(* CODESYS project pluginbeckhoffethercatasycube.library
   Author: Asyril SA
   Placeholder: Plugin Ethercat Asycube
   Title: Plugin Ethercat Asycube
   Version: 1.1.0
   Description: This library is created for controling the Asycube product
   Company: Asyril SA

Project tree, tasks and I/O mapping:
  libraries: Tc2_Standard, * (Beckhoff Automation GmbH); Tc2_System, * (Beckhoff Automation GmbH); Tc2_Utilities, * (Beckhoff Automation GmbH); Tc3_Module, * (Beckhoff Automation GmbH); VisuDialogs, * (System); VisuSymbols, 3.5.10.0 (System)
  DUTs/
    data type asycubeReadHoldingRegister
    data type asycubeWriteHoldingRegister
    data type HOLDING_REGISTERS_READ
    data type HOLDING_REGISTERS_WRITE
  GVLs/
    global variables dbGateway
  POUs/
    function block FB_Backlight [ST]
    function block FB_Execute_Hopper_Vibration [ST]
    function block FB_Execute_Platform_Vibration [ST]
    function block FB_Execute_Sequence [ST]
    program MAIN [FBD]
  VISUs/
  text list GlobalTextList
*)

// DUTs/asycubeReadHoldingRegister
TYPE asycubeReadHoldingRegister :
UNION
	w				: INT;
	b 		AT %I* 	: ARRAY[0..1] OF BYTE;
END_UNION
END_TYPE

// DUTs/asycubeWriteHoldingRegister
TYPE asycubeWriteHoldingRegister :
UNION
	w				: INT;
	b 		AT %Q* 	: ARRAY[0..1] OF BYTE;
END_UNION
END_TYPE

// DUTs/HOLDING_REGISTERS_READ
TYPE HOLDING_REGISTERS_READ :
STRUCT
	HR_MODBUS_STATUS: asycubeReadHoldingRegister;
	HR_MODBUS_ERROR_CODE: asycubeReadHoldingRegister;
	HR_WARNINGS: asycubeReadHoldingRegister;
	HR_ALARMS: asycubeReadHoldingRegister;
	HR_MODBUS_PLATFORM_STATUS: asycubeReadHoldingRegister;
	HR_PLATFORM_REMAINING_TIME: asycubeReadHoldingRegister;
	HR_MODBUS_HOPPER_STATUS: asycubeReadHoldingRegister;
	HR_HOPPER_REMAINING_TIME: asycubeReadHoldingRegister;
	HR_MODBUS_SEQUENCE_STATUS: asycubeReadHoldingRegister;
	HR_SEQUENCE_REMAINING_TIME: asycubeReadHoldingRegister;
	HR_VIBRATION_SET_SELECTED: asycubeReadHoldingRegister;
	HR_SEQUENCE_SELECTED: asycubeReadHoldingRegister;
	HR_BACKLIGHT_STATE_STATUS: asycubeReadHoldingRegister;
	HR_READ_WRITE_PARAMETER_READ_VALUE: asycubeReadHoldingRegister;
	HR_FIRMWARE_VERSION_H: asycubeReadHoldingRegister;
	HR_FIRMWARE_VERSION_M: asycubeReadHoldingRegister;
	HR_FIRMWARE_VERSION_L: asycubeReadHoldingRegister;
	HR_USER_ACCESS_LEVEL: asycubeReadHoldingRegister;
	HR_FLASH_OPERATIONS_STATUS: asycubeReadHoldingRegister;
	HR_MODBUS_COMMUNICATION_STATUS_L: asycubeReadHoldingRegister;
	HR_MODBUS_COMMUNICATION_STATUS_H: asycubeReadHoldingRegister;
	HR_ETHERCAT_COMMUNICATION_STATUS: asycubeReadHoldingRegister;

END_STRUCT
END_TYPE

// DUTs/HOLDING_REGISTERS_WRITE
TYPE HOLDING_REGISTERS_WRITE :
STRUCT
	HR_MODBUS_CONTROL: asycubeWriteHoldingRegister;
	HR_PLATFORM_VIBRATION_TRIG: asycubeWriteHoldingRegister;
	HR_PLATFORM_VIBRATION_ID: asycubeWriteHoldingRegister;
	HR_PLATFORM_VIBRATION_DURATION: asycubeWriteHoldingRegister;
	HR_PLATFORM_CENTERING_TRIG: asycubeWriteHoldingRegister;
	HR_PLATFORM_CENTERING_X: asycubeWriteHoldingRegister;
	HR_PLATFORM_CENTERING_Y: asycubeWriteHoldingRegister;
	HR_HOPPER_VIBRATION_TRIG: asycubeWriteHoldingRegister;
	HR_HOPPER_VIBRATION_ID: asycubeWriteHoldingRegister;
	HR_HOPPER_VIBRATION_DURATION: asycubeWriteHoldingRegister;
	HR_HOPPER_FEEDING_TRIG: asycubeWriteHoldingRegister;
	HR_HOPPER_FEEDING_VIBRATION: asycubeWriteHoldingRegister;
	HR_HOPPER_FEEDING_NBPARTS: asycubeWriteHoldingRegister;
	HR_HOPPER_FEEDING_NBMAX: asycubeWriteHoldingRegister;
	HR_SEQUENCE_EXECUTION_TRIG: asycubeWriteHoldingRegister;
	HR_SEQUENCE_EXECUTION_NBPARTS: asycubeWriteHoldingRegister;
	HR_SEQUENCE_EXECUTION_NBMAX: asycubeWriteHoldingRegister;
	HR_SEQUENCE_EXECUTION_X: asycubeWriteHoldingRegister;
	HR_SEQUENCE_EXECUTION_Y: asycubeWriteHoldingRegister;
	HR_SEQUENCE_EXECUTION_SEQUENCEID: asycubeWriteHoldingRegister;
	HR_SELECT_VIBRATION_SET: asycubeWriteHoldingRegister;
	HR_SELECT_SEQUENCE: asycubeWriteHoldingRegister;
	HR_BACKLIGHT_STATE_CONTROL: asycubeWriteHoldingRegister;
	HR_EXECUTE_BACKLIGHT_FLASH_TRIG: asycubeWriteHoldingRegister;
	HR_BACKLIGHT_INTENSITY_TRIG: asycubeWriteHoldingRegister;
	HR_BACKLIGHT_INTENSITY: asycubeWriteHoldingRegister;
	HR_PLATFORM_HALT: asycubeWriteHoldingRegister;
	HR_HOPPER_HALT: asycubeWriteHoldingRegister;
	HR_SEQUENCE_HALT: asycubeWriteHoldingRegister;
	HR_READ_WRITE_PARAMETER_TRIG: asycubeWriteHoldingRegister;
	HR_READ_WRITE_PARAMETER_ADDRESS: asycubeWriteHoldingRegister;
	HR_READ_WRITE_PARAMETER_WRITE_VALUE: asycubeWriteHoldingRegister;
	HR_FLASH_OPERATIONS: asycubeWriteHoldingRegister;
	
END_STRUCT
END_TYPE

// GVLs/dbGateway
{attribute 'qualified_only'}
VAR_GLOBAL
	regAsycubeRead			: HOLDING_REGISTERS_READ;		//Register for read in Asycube
	regAsycubeWrite			: HOLDING_REGISTERS_WRITE;		//Register for write in Asycube
	
END_VAR

// POUs/FB_Backlight
FUNCTION_BLOCK FB_Backlight
VAR_INPUT
	{attribute 'pingroup' := 'Working'}
	boLightONPIN				: BOOL;							//Turn ON the Backlight
	{attribute 'pingroup' := 'Working'}
	boLightOFFPIN				: BOOL;							//Turn OFF the Backlight
	{attribute 'pingroup' := 'Working'}
	tiDurationPIN				: TIME;							//Duration of backlight
	
END_VAR
VAR_IN_OUT					
	{attribute 'pingroup' := 'Gateway'}
	regAsycubeWritePIO			: HOLDING_REGISTERS_WRITE;		//Register for writing to Asycube
	{attribute 'pingroup' := 'Gateway'}
	regAsycubeReadPIO			: HOLDING_REGISTERS_READ;		//Register for reading to Asycube
	
END_VAR
VAR_OUTPUT
	{attribute 'pingroup' := 'Working'}
	woStatePOU					: WORD;							//0 = IDLE, 1 = Running, 2 = Stopping, 10 = Error
	{attribute 'pingroup' := 'Working'}
	tiRemainingTimePOU			: TIME;							//Time remaining of backlight
	
	{attribute 'pingroup' := 'Error Management'}
	boErrorPOU					: BOOL;							//Error
	{attribute 'pingroup' := 'Error Management'}
	inErrorIDPOU				: INT;							//Error ID
	{attribute 'pingroup' := 'Error Management'}
	stErrorNamePOU				: STRING;						//Name of error
	
END_VAR
VAR
	R_TRIG_Start				: R_TRIG;						//Rising edge of start
	R_TRIG_Stop					: R_TRIG;						//Rising edge of stop
	TOF_Duration				: TOF;							//Duration of backlight
	R_TRIG_State1				: R_TRIG;						//Rising edge of number sequence 1
	TON_TimeOut					: TON;							//Temporisation of time out communication
	
	woLastStateLST				: WORD;							//Last state
	boErrorTransitionLST		: BOOL;							//Error transition
	boErrorTimeOutLST			: BOOL;							//Error time out
	boErrorComAsycubeLST		: BOOL;							//Error communication Asycube
	boErrorComGatewayLST		: BOOL;							//Error communication gateway
END_VAR

//=============================================================================
// Asyril SA
// (c)Copyright 2019 
//-----------------------------------------------------------------------------
// Library:       Plugin Asycube EtherCat Beckhoff   
// Tested with:   C6015
// Engineering:   Twincat 3.1.4024.7
// Restrictions:  -
// Requirements:  -
// Functionality: FB_Backlight, Management of asycube backlight.
//-----------------------------------------------------------------------------
// Change log table:
// Version  Date       In charge / Changes applied
// 1.0      26.03.2020 DcA         Version inital.
// 1.1 		23.09.2020 DcA		   Added precision in connection errors.
// 
//=============================================================================

//Declarations of program instances (trigger and temporisation)
{region "Trigger"}

//Rising trigger of light on
R_TRIG_Start(CLK:= boLightONPIN);

//Rising trigger of light off
R_TRIG_Stop(CLK:= boLightOFFPIN);

//Rising trigger of running state
R_TRIG_State1(CLK:= woStatePOU = 1);

//Temporisation of light on
TOF_Duration(IN:= R_TRIG_State1.Q, PT:= tiDurationPIN);

//Temporisation of time out of communication
TON_TimeOut(IN:= (woStatePOU = 1 AND regAsycubeReadPIO.HR_BACKLIGHT_STATE_STATUS.w = 0)
				OR (woStatePOU = 0 AND regAsycubeReadPIO.HR_BACKLIGHT_STATE_STATUS.w = 1), PT:= T#5S);
	
//Initialisation
tiRemainingTimePOU := T#0S;		 
	 
{endregion}
	 
	 
//Region of working programm
{region "Working"}

//Sequence state diagram
CASE woStatePOU OF
	
	0:	//IDLE
	
	IF boErrorPOU THEN
		woStatePOU := 10;
	ELSIF R_TRIG_Start.Q THEN
		woStatePOU := 1;
	END_IF;
	
	1:	//Running
	
	IF boErrorPOU THEN
		woStatePOU := 10;
	ELSIF R_TRIG_Start.Q THEN
		woStatePOU := 10;
		boErrorTransitionLST := TRUE;
	ELSIF R_TRIG_Stop.Q OR (TOF_Duration.ET >= tiDurationPIN AND tiDurationPIN > T#0MS) THEN
		woStatePOU := 2;
	END_IF;
	
	2:	//Stopping
	
	IF boErrorPOU THEN
		woStatePOU := 10;
	ELSIF R_TRIG_Start.Q THEN
		woStatePOU := 10; 
		boErrorTransitionLST := TRUE;
	ELSIF regAsycubeReadPIO.HR_BACKLIGHT_STATE_STATUS.w = 0 THEN
		woStatePOU := 0;
	END_IF;
	
	10:	//Error

	IF NOT boErrorPOU THEN
		woStatePOU := 2;
	END_IF;

END_CASE;

//Parameters processing

//If it is in running
IF woStatePOU = 1 THEN
	regAsycubeWritePIO.HR_BACKLIGHT_STATE_CONTROL.w := 1;
	tiRemainingTimePOU := tiDurationPIN - TOF_Duration.ET;
END_IF;

//If it is in stopping
IF woStatePOU = 2 THEN
	regAsycubeWritePIO.HR_BACKLIGHT_STATE_CONTROL.w := 0;
	regAsycubeWritePIO.HR_MODBUS_CONTROL.w := 16#00;
END_IF;

//If it is in error
IF woStatePOU = 10 THEN
	regAsycubeWritePIO.HR_BACKLIGHT_STATE_CONTROL.w := 0;
END_IF;

//Save last state before error state
IF woStatePOU <> 10 THEN
	woLastStateLST := woStatePOU;
END_IF;

//If it is in error (trigger)
IF (R_TRIG_Stop.Q AND woStatePOU = 10) OR 
	((regAsycubeReadPIO.HR_MODBUS_COMMUNICATION_STATUS_L.w = 4 AND regAsycubeReadPIO.HR_ETHERCAT_COMMUNICATION_STATUS.w = 8) AND 
	(boErrorComAsycubeLST OR boErrorComGatewayLST) AND 
	woLastStateLST = 0) THEN
	
	regAsycubeWritePIO.HR_MODBUS_CONTROL.w := 16#FF;
	boErrorTransitionLST := FALSE;
	boErrorComAsycubeLST := FALSE;
	boErrorComGatewayLST := FALSE;
	boErrorTimeOutLST := FALSE;
END_IF;
	 
{endregion}

//Management of error
{region "Error"}
	
//Time out communciation	
IF TON_TimeOut.Q THEN
	boErrorTimeOutLST := TRUE;
END_IF;

//Asycube disconnected
IF regAsycubeReadPIO.HR_MODBUS_COMMUNICATION_STATUS_L.w <> 4 AND woStatePOU <> 10 THEN
	boErrorComAsycubeLST := TRUE;
END_IF;

//Gateway disconnected
IF regAsycubeReadPIO.HR_ETHERCAT_COMMUNICATION_STATUS.w <> 8 AND woStatePOU <> 10 THEN
	boErrorComGatewayLST := TRUE;
END_IF;
  
//If an error is active
IF	((regAsycubeReadPIO.HR_MODBUS_STATUS.w <> 0 OR boErrorTransitionLST) AND woStatePOU <> 0) OR 
	boErrorTimeOutLST OR boErrorComAsycubeLST OR boErrorComGatewayLST THEN
		 
	boErrorPOU := TRUE;
			
		//Error transition
		IF boErrorTransitionLST THEN
			inErrorIDPOU := 730;
			stErrorNamePOU := 'Transition Error';
		//Asycube  Modbus  errors  status
		ELSIF (INT_TO_UINT(regAsycubeReadPIO.HR_MODBUS_STATUS.w) AND 16#01) = 16#01 THEN	
			inErrorIDPOU := 731;	
	  		stErrorNamePOU := 'Asycube Modbus Error : 0x';
			stErrorNamePOU := CONCAT(STR1:= stErrorNamePOU, STR2:= DWORD_TO_HEXSTR( UINT_TO_DWORD( INT_TO_UINT(regAsycubeReadPIO.HR_MODBUS_ERROR_CODE.w) AND 16#00FF ), 4, FALSE ) ); 
				 
		//Internal  Modbus  communication  errorstatus
		ELSIF (INT_TO_UINT(regAsycubeReadPIO.HR_MODBUS_STATUS.w) AND 16#02) = 16#02 THEN
			inErrorIDPOU := 732;
			stErrorNamePOU := 'Asycube Internal Modbus Error : 0x';
			stErrorNamePOU := CONCAT(STR1:= stErrorNamePOU, STR2:= DWORD_TO_HEXSTR( UINT_TO_DWORD( SHL( INT_TO_UINT(regAsycubeReadPIO.HR_MODBUS_ERROR_CODE.w) AND 16#FF00 , 2) ) , 4, FALSE ) ); 
						   
		//Asycube  warnings  status
		ELSIF (INT_TO_UINT(regAsycubeReadPIO.HR_MODBUS_STATUS.w) AND 16#04) = 16#04 THEN
			inErrorIDPOU := 733;
			stErrorNamePOU := 'Asycube Warnings : 0x';
			stErrorNamePOU := CONCAT(STR1:= stErrorNamePOU, STR2:= DWORD_TO_HEXSTR( INT_TO_DWORD(regAsycubeReadPIO.HR_WARNINGS.w), 4, FALSE ) ); 

		//Asycube alarms status
		ELSIF (INT_TO_UINT(regAsycubeReadPIO.HR_MODBUS_STATUS.w) AND 16#08) = 16#08 THEN
			inErrorIDPOU := 734;
			stErrorNamePOU := 'Asycube Alarms : 0x';
			stErrorNamePOU := CONCAT(STR1:= stErrorNamePOU, STR2:= DWORD_TO_HEXSTR( INT_TO_DWORD(regAsycubeReadPIO.HR_ALARMS.w), 4, FALSE ) );   	
 
		//Gateway disconnected from plc
		ELSIF boErrorComGatewayLST THEN
			inErrorIDPOU := 735;
			stErrorNamePOU := 'Gateway disconnected from PLC';
		
		//Asycube disconnected from gateway
		ELSIF boErrorComAsycubeLST THEN
			inErrorIDPOU := 736;
			stErrorNamePOU := 'Asycube disconnected from gateway';
		
		//Communication time out
		ELSIF boErrorTimeOutLST THEN
			inErrorIDPOU := 737;
			stErrorNamePOU := 'Time out';

	 	//Unknown error
		ELSE 
			inErrorIDPOU := 739;
			stErrorNamePOU := 'N/A';
		END_IF;  

ELSE
	boErrorPOU := FALSE;
	inErrorIDPOU := 0;
	stErrorNamePOU := '';	 
END_IF;
	 
{endregion}

END_FUNCTION_BLOCK

// POUs/FB_Execute_Hopper_Vibration
FUNCTION_BLOCK FB_Execute_Hopper_Vibration
VAR_INPUT
	{attribute 'pingroup' := 'Working'}
	inSelectModePIN				: INT;							//0 = Vibration, 1 = Hopping
	{attribute 'pingroup' := 'Working'}
	boStartPIN					: BOOL;							//Start vibration
	{attribute 'pingroup' := 'Working'}
	boStopPIN					: BOOL;							//Stop vibration
	{attribute 'pingroup' := 'Working'}
	inVibrationIDPIN			: INT:=0;						//Vibration ID (0..25)
	{attribute 'pingroup' := 'Working'}
	inVibrationSetPIN			: INT:=1;						//Vibration Set (1..26)
	{attribute 'pingroup' := 'Working'}
	inNbPartsPIN				: INT;							//Number of parts on the cube
	{attribute 'pingroup' := 'Working'}
	inNbPartsMaxPIN				: INT;							//Number max of parts on the cube
	{attribute 'pingroup' := 'Working'}
	tiDurationPIN				: TIME;							//Time duration of vibration

END_VAR
VAR_IN_OUT
	{attribute 'pingroup' := 'Gateway'}
	regAsycubeWritePIO			: HOLDING_REGISTERS_WRITE;		//Register for writing to Asycube
	{attribute 'pingroup' := 'Gateway'}
	regAsycubeReadPIO			: HOLDING_REGISTERS_READ;		//Register for reading to Asycube
	
END_VAR
VAR_OUTPUT
	{attribute 'pingroup' := 'Working'}
	woStatePOU					: WORD;							//0 = IDLE, 1 = Running, 2 = Stopping, 10 = Error
	{attribute 'pingroup' := 'Working'}
	boDonePOU					: BOOL;							//Vibration is done
	{attribute 'pingroup' := 'Working'}
	tiRemainingTimePOU			: TIME;							//Time remaining of vibration
	
	{attribute 'pingroup' := 'Error Management'}
	boErrorPOU					: BOOL;							//Error
	{attribute 'pingroup' := 'Error Management'}
	inErrorIDPOU				: INT;							//Error ID
	{attribute 'pingroup' := 'Error Management'}
	stErrorNamePOU				: STRING;						//Name of error
	

END_VAR
VAR
	R_TRIG_Start				: R_TRIG;						//Rising edge of start
	R_TRIG_Stop					: R_TRIG;						//Rising edge of stop
	R_TRIG_State1				: R_TRIG;						//Rising edge step number 1
	R_TRIG_Done					: R_TRIG;						//Rising edge of vibration done 
	TON_TimeOut					: TON;							//Temporisation of time out communication
	
	woLastStateLST				: WORD;							//Last state
	boErrorTransitionLST		: BOOL;							//Error transition
	boErrorTimeOutLST			: BOOL;							//Error time out
	boErrorComAsycubeLST		: BOOL;							//Error communication Asycube
	boErrorComGatewayLST		: BOOL;							//Error communication gateway
	boErrorParameterLST			: BOOL;							//Error parameters
	
END_VAR

//=============================================================================
// Asyril SA
// (c)Copyright 2019 
//-----------------------------------------------------------------------------
// Library:       Plugin Asycube EtherCat Beckhoff   
// Tested with:   C6015
// Engineering:   Twincat 3.1.4024.7
// Restrictions:  -
// Requirements:  -
// Functionality: FB_Execute_Hopper_Vibration, Management of hopper vibration.
//-----------------------------------------------------------------------------
// Change log table:
// Version  Date       In charge / Changes applied
// 1.0      26.03.2020 DcA         Version initale.
// 1.1 		23.09.2020 DcA		   Added precision in connection errors.
// 
//=============================================================================

//Declarations of program instances (trigger and temporisation)
{region "Trigger"}

//Rising trigger of start
R_TRIG_Start(CLK:= boStartPIN);

//Rising trigger of stop
R_TRIG_Stop(CLK:= boStopPIN);

//Rising trigger of running state
R_TRIG_State1(CLK:= woStatePOU = 1);

//Rising trigger of vibration done
R_TRIG_Done(CLK:= regAsycubeReadPIO.HR_MODBUS_HOPPER_STATUS.w = 0);
	 
//Temporisation of time out of communication
TON_TimeOut(IN:= (woStatePOU = 1 AND regAsycubeReadPIO.HR_MODBUS_HOPPER_STATUS.w = 0)
				OR (woStatePOU = 0 AND regAsycubeReadPIO.HR_MODBUS_HOPPER_STATUS.w = 1), PT:= T#5S);
		  
{endregion}
	 
//Region of working programm
{region "Working"}

//Sequence state diagram
CASE woStatePOU OF
	
	0:	//IDLE
		 
	IF boErrorPOU THEN
		woStatePOU := 10;
		boDonePOU := FALSE;
	ELSIF R_TRIG_Start.Q THEN
		woStatePOU := 1;
		boDonePOU := FALSE;
	END_IF;
	
	1:	//Running

	IF boErrorPOU THEN
		woStatePOU := 10;
	ELSIF R_TRIG_Start.Q THEN
		woStatePOU := 10;
		boErrorTransitionLST := TRUE;
	ELSIF R_TRIG_Stop.Q THEN
		woStatePOU := 2;
	ELSIF R_TRIG_Done.Q THEN
		woStatePOU := 2;
		boDonePOU := TRUE;
	END_IF;
	
	2:	//Stopping

	IF boErrorPOU THEN
		woStatePOU := 10;
	ELSIF R_TRIG_Start.Q THEN
		woStatePOU := 10;
		boErrorTransitionLST := TRUE;
	ELSIF regAsycubeReadPIO.HR_MODBUS_HOPPER_STATUS.w = 0 THEN
		woStatePOU := 0;
	END_IF;
	
	10:	//Error

	IF NOT boErrorPOU THEN
		woStatePOU := 2;
	END_IF;

END_CASE;

//Parameters processing

//If it is in IDLE
IF woStatePOU = 0 THEN
	regAsycubeWritePIO.HR_HOPPER_HALT.w := 0;
END_IF;

//If it is in running (trigger) and vibration mode
IF R_TRIG_State1.Q AND inSelectModePIN = 0 THEN
	regAsycubeWritePIO.HR_HOPPER_VIBRATION_TRIG.w := 1;
END_IF;

//If it is in running (trigger) and feeding mode
IF R_TRIG_State1.Q AND inSelectModePIN = 1 THEN
	regAsycubeWritePIO.HR_HOPPER_FEEDING_TRIG.w := 1;
END_IF;

//If it is in running
IF inSelectModePIN = 0 AND tiDurationPIN = T#0MS THEN
	tiRemainingTimePOU := T#0S;
ELSE
	tiRemainingTimePOU := INT_TO_TIME(regAsycubeReadPIO.HR_HOPPER_REMAINING_TIME.w);
END_IF;

//If it is in stopping
IF woStatePOU = 2 THEN
	regAsycubeWritePIO.HR_HOPPER_VIBRATION_TRIG.w := 0;
	regAsycubeWritePIO.HR_HOPPER_FEEDING_TRIG.w := 0;
	regAsycubeWritePIO.HR_HOPPER_HALT.w := 1;
	regAsycubeWritePIO.HR_MODBUS_CONTROL.w := 16#00;
END_IF;

//If it is in error
IF woStatePOU = 10 THEN
	regAsycubeWritePIO.HR_HOPPER_VIBRATION_TRIG.w := 0;
	regAsycubeWritePIO.HR_HOPPER_FEEDING_TRIG.w := 0;
	regAsycubeWritePIO.HR_HOPPER_HALT.w := 1;
END_IF;
		  
//Save last state before error state
IF woStatePOU <> 10 THEN
	woLastStateLST := woStatePOU;
END_IF;

//If it is in error (trigger)
IF (R_TRIG_Stop.Q AND woStatePOU = 10) OR 
	((regAsycubeReadPIO.HR_MODBUS_COMMUNICATION_STATUS_L.w = 4 AND regAsycubeReadPIO.HR_ETHERCAT_COMMUNICATION_STATUS.w = 8) AND 
	(boErrorComAsycubeLST OR boErrorComGatewayLST) AND 
	woLastStateLST = 0) THEN
	
	regAsycubeWritePIO.HR_MODBUS_CONTROL.w := 16#FF;
	boErrorTransitionLST := FALSE;
	boErrorTimeOutLST := FALSE;
	boErrorComAsycubeLST := FALSE;
	boErrorComGatewayLST := FALSE;
	boErrorParameterLST := FALSE;
END_IF;

//Set parameters
//Position and duration paramater
regAsycubeWritePIO.HR_HOPPER_VIBRATION_DURATION.w := TIME_TO_INT(tiDurationPIN);
regAsycubeWritePIO.HR_HOPPER_FEEDING_NBMAX.w := inNbPartsMaxPIN;
regAsycubeWritePIO.HR_HOPPER_FEEDING_NBPARTS.w := inNbPartsPIN;

//Vibration ID parameter
IF inVibrationIDPIN > 25 AND woStatePOU = 1 THEN
	boErrorParameterLST := TRUE;
ELSIF inVibrationIDPIN < 0 AND woStatePOU = 1 THEN
	boErrorParameterLST := TRUE;
ELSIF woStatePOU = 1 THEN
	regAsycubeWritePIO.HR_HOPPER_VIBRATION_ID.w := inVibrationIDPIN;
	regAsycubeWritePIO.HR_HOPPER_FEEDING_VIBRATION.w := inVibrationIDPIN;
END_IF;

//Vibration set parameter  
IF inVibrationSetPIN > 26 AND woStatePOU = 1 THEN
	boErrorParameterLST := TRUE;
ELSIF inVibrationSetPIN < 1 AND woStatePOU = 1 THEN
	boErrorParameterLST := TRUE;
ELSIF woStatePOU = 1 THEN
	regAsycubeWritePIO.HR_SELECT_VIBRATION_SET.w := inVibrationSetPIN;
END_IF;

{endregion}

//Reion Error management
{region "Error"}

//Time out communication
IF TON_TimeOut.Q THEN
	boErrorTimeOutLST := TRUE;
END_IF;

//Asycube disconnected
IF regAsycubeReadPIO.HR_MODBUS_COMMUNICATION_STATUS_L.w <> 4 AND woStatePOU <> 10 THEN
	boErrorComAsycubeLST := TRUE;
END_IF;

//Gateway disconnected
IF regAsycubeReadPIO.HR_ETHERCAT_COMMUNICATION_STATUS.w <> 8 AND woStatePOU <> 10 THEN
	boErrorComGatewayLST := TRUE;
END_IF;

//If an error is active
IF	((regAsycubeReadPIO.HR_MODBUS_STATUS.w <> 0 OR boErrorTransitionLST OR boErrorParameterLST) AND woStatePOU <> 0) OR 
	boErrorTimeOutLST OR boErrorComAsycubeLST OR 
	boErrorComGatewayLST OR regAsycubeReadPIO.HR_MODBUS_HOPPER_STATUS.w = 2 THEN
	
	boErrorPOU := TRUE;
			
		//Error transition
		IF boErrorTransitionLST THEN
			inErrorIDPOU := 720;
			stErrorNamePOU := 'Transition Error';
		//Asycube  Modbus  errors  status
		ELSIF (INT_TO_UINT(regAsycubeReadPIO.HR_MODBUS_STATUS.w) AND 16#01) = 16#01 THEN	
			inErrorIDPOU := 721;	
	  		stErrorNamePOU := 'Asycube Modbus Error : 0x';
			stErrorNamePOU := CONCAT(STR1:= stErrorNamePOU, STR2:= DWORD_TO_HEXSTR( UINT_TO_DWORD( INT_TO_UINT(regAsycubeReadPIO.HR_MODBUS_ERROR_CODE.w) AND 16#00FF ), 4, FALSE ) ); 
				 
		//Internal  Modbus  communication  errorstatus
		ELSIF (INT_TO_UINT(regAsycubeReadPIO.HR_MODBUS_STATUS.w) AND 16#02) = 16#02 THEN
			inErrorIDPOU := 722;
			stErrorNamePOU := 'Asycube Internal Modbus Error : 0x';
			stErrorNamePOU := CONCAT(STR1:= stErrorNamePOU, STR2:= DWORD_TO_HEXSTR( UINT_TO_DWORD( SHL( INT_TO_UINT(regAsycubeReadPIO.HR_MODBUS_ERROR_CODE.w) AND 16#FF00 , 2) ) , 4, FALSE ) ); 
						   
		//Asycube  warnings  status
		ELSIF (INT_TO_UINT(regAsycubeReadPIO.HR_MODBUS_STATUS.w) AND 16#04) = 16#04 THEN
			inErrorIDPOU := 723;
			stErrorNamePOU := 'Asycube Warnings : 0x';
			stErrorNamePOU := CONCAT(STR1:= stErrorNamePOU, STR2:= DWORD_TO_HEXSTR( INT_TO_DWORD(regAsycubeReadPIO.HR_WARNINGS.w), 4, FALSE ) ); 

		//Asycube alarms status
		ELSIF (INT_TO_UINT(regAsycubeReadPIO.HR_MODBUS_STATUS.w) AND 16#08) = 16#08 THEN
			inErrorIDPOU := 724;
			stErrorNamePOU := 'Asycube Alarms : 0x';
			stErrorNamePOU := CONCAT(STR1:= stErrorNamePOU, STR2:= DWORD_TO_HEXSTR( INT_TO_DWORD(regAsycubeReadPIO.HR_ALARMS.w), 4, FALSE ) );   	
 
		//Gateway disconnected from plc
		ELSIF boErrorComGatewayLST THEN
			inErrorIDPOU := 725;
			stErrorNamePOU := 'Gateway disconnected from PLC';
		
		//Asycube disconnected from gateway
		ELSIF boErrorComAsycubeLST THEN
			inErrorIDPOU := 726;
			stErrorNamePOU := 'Asycube disconnected from gateway';
		
		//Communication time out
		ELSIF boErrorTimeOutLST THEN
			inErrorIDPOU := 727;
			stErrorNamePOU := 'Time out';
			 
		//Incorrect parameters
		ELSIF boErrorParameterLST THEN
			inErrorIDPOU := 728;
			stErrorNamePOU := 'Wrong parameter';
			//See variable error
			IF inVibrationIDPIN > 26 OR inVibrationIDPIN < 1 THEN
				stErrorNamePOU := CONCAT(stErrorNamePOU , ' : inVibrationIDPIN' );
			ELSIF inVibrationSetPIN > 26 OR inVibrationSetPIN < 1 THEN
				stErrorNamePOU := CONCAT(stErrorNamePOU , ' : inVibrationSetPIN' );
			END_IF;
				 
		//Unknown error
		ELSE 
			inErrorIDPOU := 729;
			stErrorNamePOU := 'N/A';
		END_IF;  

ELSE
	boErrorPOU := FALSE;
	inErrorIDPOU := 0;
	stErrorNamePOU := '';	 
END_IF;
	 
{endregion}

END_FUNCTION_BLOCK

// POUs/FB_Execute_Platform_Vibration
FUNCTION_BLOCK FB_Execute_Platform_Vibration
VAR_INPUT
	{attribute 'pingroup' := 'Working'}
	inSelectModePIN				: INT;							//0 = Vibration, 1 = Centering
	{attribute 'pingroup' := 'Working'}
	boStartPIN					: BOOL;							//Start vibration
	{attribute 'pingroup' := 'Working'}
	boStopPIN					: BOOL;							//Stop vibration
	{attribute 'pingroup' := 'Working'}
	inVibrationIDPIN			: INT:=0;						//Vibration ID (0..25)
	{attribute 'pingroup' := 'Working'}
	inVibrationSetPIN			: INT:=1;						//Vibration Set (1..26)
	{attribute 'pingroup' := 'Working'}
	inXPosPIN					: INT;							//Global part in position X (-100, 0, 100)
	{attribute 'pingroup' := 'Working'}
	inYPosPIN					: INT;							//Global part in position Y (-100, 0, 100)
	{attribute 'pingroup' := 'Working'}
	tiDurationPIN				: TIME;							//Time remaining vibration

END_VAR
VAR_IN_OUT
	{attribute 'pingroup' := 'Gateway'}
	regAsycubeWritePIO			: HOLDING_REGISTERS_WRITE;		//Register for writing to Asycube
	{attribute 'pingroup' := 'Gateway'}
	regAsycubeReadPIO			: HOLDING_REGISTERS_READ;		//Register for reading to Asycube
	
END_VAR
VAR_OUTPUT
	{attribute 'pingroup' := 'Working'}
	woStatePOU					: WORD;							//0 = IDLE, 1 = Running, 2 = Stopping, 10 = Error
	{attribute 'pingroup' := 'Working'}
	boDonePOU					: BOOL;							//Vibration is done
	{attribute 'pingroup' := 'Working'}
	tiRemainingTimePOU			: TIME;							//Time remaining
	
	{attribute 'pingroup' := 'Error Management'}
	boErrorPOU					: BOOL;							//Error
	{attribute 'pingroup' := 'Error Management'}
	inErrorIDPOU				: INT;							//Error ID
	{attribute 'pingroup' := 'Error Management'}
	stErrorNamePOU				: STRING;						//Name of error

END_VAR
VAR
	R_TRIG_Start				: R_TRIG;						//Rising edge of start
	R_TRIG_Stop					: R_TRIG;						//Rising edge of stop
	R_TRIG_State1				: R_TRIG;						//Rising edge step number 1
	R_TRIG_Done					: R_TRIG;						//Rising edge of vibration done
	TON_TimeOut					: TON;							//Temporisation of time out communication
	
	woLastStateLST				: WORD;							//Last state
	boErrorTransitionLST		: BOOL;							//Error transition
	boErrorTimeOutLST			: BOOL;							//Error time out
	boErrorComAsycubeLST		: BOOL;							//Error communication Asycube
	boErrorComGatewayLST		: BOOL;							//Error communication gateway
	boErrorParameterLST			: BOOL;							//Error parameters
	
END_VAR

//=============================================================================
// Asyril SA
// (c)Copyright 2019 
//-----------------------------------------------------------------------------
// Library:       Plugin Asycube EtherCat Beckhoff   
// Tested with:   C6015
// Engineering:   Twincat 3.1.4024.7
// Restrictions:  -
// Requirements:  -
// Functionality: FB_Execute_Platform_Vibration, Management of platform vibration.
//-----------------------------------------------------------------------------
// Change log table:
// Version  Date       In charge / Changes applied
// 1.0      26.03.2020 DcA         Version initale.
// 1.1 		23.09.2020 DcA		   Added precision in connection errors.
// 
//=============================================================================

//Declarations of program instances (trigger and temporisation)
{region "Trigger"}

//Rising trigger of start
R_TRIG_Start(CLK:= boStartPIN);

//Rising trigger of stop
R_TRIG_Stop(CLK:= boStopPIN);

//Rising trigger of running state
R_TRIG_State1(CLK:= woStatePOU = 1);

//Rising trigger of running state
R_TRIG_Done(CLK:= regAsycubeReadPIO.HR_MODBUS_PLATFORM_STATUS.w = 0);

//Temporisation of time out of communication
TON_TimeOut(IN:= (woStatePOU = 1 AND regAsycubeReadPIO.HR_MODBUS_PLATFORM_STATUS.w = 0)
				OR (woStatePOU = 0 AND regAsycubeReadPIO.HR_MODBUS_PLATFORM_STATUS.w = 1), PT:= T#5S);

{endregion}
	 
//Region of working programm
{region "Working"}

//Sequence state diagram
CASE woStatePOU OF
	
	0:	//IDLE

	IF boErrorPOU THEN
		woStatePOU := 10;
		boDonePOU := FALSE;
	ELSIF R_TRIG_Start.Q THEN
		woStatePOU := 1;
		boDonePOU := FALSE;
	END_IF;
	
	1:	//Running

	IF boErrorPOU THEN
		woStatePOU := 10;
	ELSIF R_TRIG_Start.Q THEN
		woStatePOU := 10;
		boErrorTransitionLST := TRUE;
	ELSIF R_TRIG_Stop.Q THEN
		woStatePOU := 2;
	ELSIF R_TRIG_Done.Q THEN
		woStatePOU := 2;
		boDonePOU := TRUE;
	END_IF;
	
	2:	//Stopping

	IF boErrorPOU THEN
		woStatePOU := 10;
	ELSIF R_TRIG_Start.Q THEN
		woStatePOU := 10;
		boErrorTransitionLST := TRUE;
	ELSIF regAsycubeReadPIO.HR_MODBUS_PLATFORM_STATUS.w = 0 THEN
		woStatePOU := 0;
	END_IF;
	
	10:	//Error

	IF NOT boErrorPOU THEN
		woStatePOU := 2;
	END_IF;

END_CASE;

//Parameters processing

//If it is in IDLE
IF woStatePOU = 0 THEN
	regAsycubeWritePIO.HR_PLATFORM_HALT.w := 0;
END_IF;

//If it is in running (trigger) and vibration mode
IF R_TRIG_State1.Q AND inSelectModePIN = 0 THEN
	regAsycubeWritePIO.HR_PLATFORM_VIBRATION_DURATION.w := TIME_TO_INT(tiDurationPIN);
	regAsycubeWritePIO.HR_PLATFORM_VIBRATION_TRIG.w:=1;
END_IF;

//If it is in running (trigger) and centering mode
IF R_TRIG_State1.Q AND inSelectModePIN = 1 THEN
	regAsycubeWritePIO.HR_PLATFORM_CENTERING_TRIG.w:=1;
END_IF;

//If it is in running (trigger)
IF inSelectModePIN = 0 AND tiDurationPIN = T#0S THEN
	tiRemainingTimePOU := T#0S;
ELSE
	tiRemainingTimePOU := INT_TO_TIME(regAsycubeReadPIO.HR_PLATFORM_REMAINING_TIME.w);
END_IF;

//If it is in stopping
IF woStatePOU = 2 THEN
	regAsycubeWritePIO.HR_PLATFORM_VIBRATION_TRIG.w:=0;
	regAsycubeWritePIO.HR_PLATFORM_CENTERING_TRIG.w:=0;
	regAsycubeWritePIO.HR_PLATFORM_HALT.w := 1;
	regAsycubeWritePIO.HR_MODBUS_CONTROL.w := 16#00;
END_IF;

//If it is in error
IF woStatePOU = 10 THEN
	regAsycubeWritePIO.HR_PLATFORM_VIBRATION_TRIG.w:=0;
	regAsycubeWritePIO.HR_PLATFORM_CENTERING_TRIG.w:=0;
	regAsycubeWritePIO.HR_PLATFORM_HALT.w := 1;
END_IF;

//Save last state before error state
IF woStatePOU <> 10 THEN
	woLastStateLST := woStatePOU;
END_IF;

//If it is in error (trigger)
IF (R_TRIG_Stop.Q AND woStatePOU = 10) OR 
	((regAsycubeReadPIO.HR_MODBUS_COMMUNICATION_STATUS_L.w = 4 AND regAsycubeReadPIO.HR_ETHERCAT_COMMUNICATION_STATUS.w = 8) AND 
	(boErrorComAsycubeLST OR boErrorComGatewayLST) AND 
	woLastStateLST = 0) THEN
	
	regAsycubeWritePIO.HR_MODBUS_CONTROL.w := 16#FF;
	boErrorTransitionLST := FALSE;
	boErrorTimeOutLST := FALSE;
	boErrorComAsycubeLST := FALSE;
	boErrorComGatewayLST := FALSE;
	boErrorParameterLST := FALSE;
END_IF;
	 
//Position X
IF inXPosPIN > 100 AND woStatePOU = 1 THEN
	boErrorParameterLST := TRUE;
ELSIF inXPosPIN < -100 AND woStatePOU = 1 THEN
	boErrorParameterLST := TRUE;
ELSIF woStatePOU = 1 THEN
	regAsycubeWritePIO.HR_PLATFORM_CENTERING_X.w:= inXPosPIN;
END_IF;

//Position Y
IF inYPosPIN > 100 AND woStatePOU = 1 THEN
	boErrorParameterLST := TRUE;
ELSIF inYPosPIN < -100 AND woStatePOU = 1 THEN
	boErrorParameterLST := TRUE;
ELSIF woStatePOU = 1 THEN
	regAsycubeWritePIO.HR_PLATFORM_CENTERING_Y.w:= inYPosPIN;
END_IF;

//Vibration set
IF inVibrationSetPIN > 26 AND woStatePOU = 1 THEN
	boErrorParameterLST := TRUE;
ELSIF inVibrationSetPIN < 1 AND woStatePOU = 1 THEN
	boErrorParameterLST := TRUE;
ELSIF woStatePOU = 1 THEN
	regAsycubeWritePIO.HR_SELECT_VIBRATION_SET.w := inVibrationSetPIN;
END_IF;

//Vibration ID parameters
IF inVibrationIDPIN > 25 AND woStatePOU = 1 THEN
	boErrorParameterLST := TRUE;
ELSIF inVibrationIDPIN < 0 AND woStatePOU = 1 THEN
	boErrorParameterLST := TRUE;
ELSIF woStatePOU = 1 THEN
	regAsycubeWritePIO.HR_PLATFORM_VIBRATION_ID.w := inVibrationIDPIN; 
END_IF;	

{endregion}

//Management of error
{region "Error"}

//Time out communciation	
IF TON_TimeOut.Q THEN
	boErrorTimeOutLST := TRUE;
END_IF;

//Asycube disconnected
IF regAsycubeReadPIO.HR_MODBUS_COMMUNICATION_STATUS_L.w <> 4 AND woStatePOU <> 10 THEN
	boErrorComAsycubeLST := TRUE;
END_IF;

//Gateway disconnected
IF regAsycubeReadPIO.HR_ETHERCAT_COMMUNICATION_STATUS.w <> 8 AND woStatePOU <> 10 THEN
	boErrorComGatewayLST := TRUE;
END_IF;
  
//If an error is active
IF	((regAsycubeReadPIO.HR_MODBUS_STATUS.w <> 0 OR boErrorTransitionLST OR
	boErrorParameterLST) AND woStatePOU <> 0) OR boErrorTimeOutLST OR boErrorComAsycubeLST OR 
	boErrorComGatewayLST OR regAsycubeReadPIO.HR_MODBUS_PLATFORM_STATUS.w = 2 THEN
		 
	boErrorPOU := TRUE;
			
		//Error transition
		IF boErrorTransitionLST THEN
			inErrorIDPOU := 710;
			stErrorNamePOU := 'Transition Error';
		//Asycube  Modbus  errors  status
		ELSIF (INT_TO_UINT(regAsycubeReadPIO.HR_MODBUS_STATUS.w) AND 16#01) = 16#01 THEN	
			inErrorIDPOU := 711;	
	  		stErrorNamePOU := 'Asycube Modbus Error : 0x';
			stErrorNamePOU := CONCAT(STR1:= stErrorNamePOU, STR2:= DWORD_TO_HEXSTR( UINT_TO_DWORD( INT_TO_UINT(regAsycubeReadPIO.HR_MODBUS_ERROR_CODE.w) AND 16#00FF ), 4, FALSE ) ); 
				 
		//Internal  Modbus  communication  errorstatus
		ELSIF (INT_TO_UINT(regAsycubeReadPIO.HR_MODBUS_STATUS.w) AND 16#02) = 16#02 THEN
			inErrorIDPOU := 712;
			stErrorNamePOU := 'Asycube Internal Modbus Error : 0x';
			stErrorNamePOU := CONCAT(STR1:= stErrorNamePOU, STR2:= DWORD_TO_HEXSTR( UINT_TO_DWORD( SHL( INT_TO_UINT(regAsycubeReadPIO.HR_MODBUS_ERROR_CODE.w) AND 16#FF00 , 2) ) , 4, FALSE ) ); 
						   
		//Asycube  warnings  status
		ELSIF (INT_TO_UINT(regAsycubeReadPIO.HR_MODBUS_STATUS.w) AND 16#04) = 16#04 THEN
			inErrorIDPOU := 713;
			stErrorNamePOU := 'Asycube Warnings : 0x';
			stErrorNamePOU := CONCAT(STR1:= stErrorNamePOU, STR2:= DWORD_TO_HEXSTR( INT_TO_DWORD(regAsycubeReadPIO.HR_WARNINGS.w), 4, FALSE ) ); 

		//Asycube alarms status
		ELSIF (INT_TO_UINT(regAsycubeReadPIO.HR_MODBUS_STATUS.w) AND 16#08) = 16#08 THEN
			inErrorIDPOU := 714;
			stErrorNamePOU := 'Asycube Alarms : 0x';
			stErrorNamePOU := CONCAT(STR1:= stErrorNamePOU, STR2:= DWORD_TO_HEXSTR( INT_TO_DWORD(regAsycubeReadPIO.HR_ALARMS.w), 4, FALSE ) );   	
 
		//Gateway disconnected from plc
		ELSIF boErrorComGatewayLST THEN
			inErrorIDPOU := 715;
			stErrorNamePOU := 'Gateway disconnected from PLC';
		
		//Asycube disconnected from gateway
		ELSIF boErrorComAsycubeLST THEN
			inErrorIDPOU := 716;
			stErrorNamePOU := 'Asycube disconnected from gateway';
		
		//Communication time out
		ELSIF boErrorTimeOutLST THEN
			inErrorIDPOU := 717;
			stErrorNamePOU := 'Time out';
		
		//Incorrect parameters
		ELSIF boErrorParameterLST THEN
			inErrorIDPOU := 718;
			stErrorNamePOU := 'Wrong parameter';
			//See variable error
			IF inXPosPIN > 100 OR inXPosPIN < -100 THEN
				stErrorNamePOU := CONCAT(stErrorNamePOU , ' : inXPosPIN' );
			ELSIF inYPosPIN > 100 OR inYPosPIN < -100 THEN
				stErrorNamePOU := CONCAT(stErrorNamePOU , ' : inYPosPIN' );
			ELSIF inVibrationIDPIN > 26 OR inVibrationIDPIN < 1 THEN
				stErrorNamePOU := CONCAT(stErrorNamePOU , ' : inVibrationIDPIN' );
			ELSIF inVibrationSetPIN > 26 OR inVibrationSetPIN < 1 THEN
				stErrorNamePOU := CONCAT(stErrorNamePOU , ' : inVibrationSetPIN' );
			END_IF;
			
		//Unknown error	 
		ELSE 
			inErrorIDPOU := 719;
			stErrorNamePOU := 'N/A';
		END_IF;  

ELSE
	boErrorPOU := FALSE;
	inErrorIDPOU := 0;
	stErrorNamePOU := '';	 
END_IF;

{endregion}

END_FUNCTION_BLOCK

// POUs/FB_Execute_Sequence
FUNCTION_BLOCK FB_Execute_Sequence
VAR_INPUT
	{attribute 'pingroup' := 'Working'}
	boStartPIN					: BOOL;							//Start sequence
	{attribute 'pingroup' := 'Working'}
	boStopPIN					: BOOL;							//Stop sequence
	{attribute 'pingroup' := 'Working'}
	inSeqIDPIN					: INT:=1;						//Sequence ID (1..26)
	{attribute 'pingroup' := 'Working'}
	inVibrationSetPIN			: INT:=1;						//Vibration Set (1..26)
	{attribute 'pingroup' := 'Working'}
	inNbPartsPIN				: INT;							//Number of parts on the cube
	{attribute 'pingroup' := 'Working'}
	inNbPartsMaxPIN				: INT;							//Number max of parts on the cube
	{attribute 'pingroup' := 'Working'}
	inXPosPIN					: INT;							//Global part in position X (-100, 0, 100)
	{attribute 'pingroup' := 'Working'}
	inYPosPIN					: INT;							//Global part in position Y (-100, 0, 100)
	{attribute 'pingroup' := 'Working'}
	boBacklightPIN				: BOOL;							//Turn ON the backlight
	
END_VAR
VAR_IN_OUT
	{attribute 'pingroup' := 'Gateway'}
	regAsycubeWritePIO			: HOLDING_REGISTERS_WRITE;		//Register for writing to Asycube
	{attribute 'pingroup' := 'Gateway'}
	regAsycubeReadPIO			: HOLDING_REGISTERS_READ;		//Register for reading to Asycube
	
END_VAR
VAR_OUTPUT
	{attribute 'pingroup' := 'Working'}
	woStatePOU					: WORD;							//0 = IDLE, 1 = Running, 2 = Stopping, 10 = Error
	{attribute 'pingroup' := 'Working'}
	boDonePOU					: BOOL;							//Sequence done
	{attribute 'pingroup' := 'Working'}
	boBacklightStatePOU			: BOOL;							//Backlight turned on
	
	{attribute 'pingroup' := 'Working'}
	tiRemainingTimePOU			: TIME;							//Time remaining
	
	{attribute 'pingroup' := 'Error Management'}
	boErrorPOU					: BOOL;							//Error
	{attribute 'pingroup' := 'Error Management'}
	inErrorIDPOU				: INT;							//Error ID
	{attribute 'pingroup' := 'Error Management'}
	stErrorNamePOU				: STRING;						//Name of error
	
END_VAR

VAR
	R_TRIG_Start				: R_TRIG;						//Rising edge of start
	R_TRIG_Stop					: R_TRIG;						//Rising edge of stop
	R_TRIG_State1				: R_TRIG;						//Rising edge step number 1
	R_TRIG_Done					: R_TRIG;						//Rising edge of sequence done
	TON_TimeOut					: TON;							//Temporisation of time out communication
	
	woLastStateLST				: WORD;							//Last state
	boErrorTransitionLST		: BOOL;							//Error transition
	boErrorTimeOutLST			: BOOL;							//Error time out
	boErrorComAsycubeLST		: BOOL;							//Error communication Asycube
	boErrorComGatewayLST		: BOOL;							//Error communication gateway
	boErrorParameterLST			: BOOL;							//Error parameters
	
END_VAR

//=============================================================================
// Asyril SA
// (c)Copyright 2019 
//-----------------------------------------------------------------------------
// Library:       Plugin Asycube EtherCat Beckhoff   
// Tested with:   C6015
// Engineering:   Twincat 3.1.4024.7
// Restrictions:  -
// Requirements:  -
// Functionality: FB_Execute_Sequence, Management of sequence vibration.
//-----------------------------------------------------------------------------
// Change log table:
// Version  Date       In charge / Changes applied
// 1.0      26.03.2020 DcA         Version initale.
// 1.1 		23.09.2020 DcA		   Added precision in connection errors.
// 
//=============================================================================

//Declarations of program instances (trigger and temporisation)
{region "Trigger"}

//Rising trigger of start
R_TRIG_Start(CLK:= boStartPIN);

//Rising trigger of stop
R_TRIG_Stop(CLK:= boStopPIN);

//Rising trigger of running state
R_TRIG_State1(CLK:= woStatePOU = 1);
	 
//Rising trigger of sequence done
R_TRIG_Done(CLK:= regAsycubeReadPIO.HR_MODBUS_SEQUENCE_STATUS.w = 0);
	 
//Temporisation time out of communication
TON_TimeOut(IN:= (woStatePOU = 1 AND regAsycubeReadPIO.HR_MODBUS_SEQUENCE_STATUS.w = 0)
				OR (woStatePOU = 0 AND regAsycubeReadPIO.HR_MODBUS_SEQUENCE_STATUS.w = 1) OR 
				(boBacklightPIN AND regAsycubeReadPIO.HR_BACKLIGHT_STATE_STATUS.w = 0)
				OR (NOT boBacklightPIN AND regAsycubeReadPIO.HR_BACKLIGHT_STATE_STATUS.w = 1), PT:= T#5S);
	 
{endregion}
	 
//Region of working programm
{region "Working"}

//Sequence state diagram
CASE woStatePOU OF
	
	0:	//IDLE

	IF boErrorPOU THEN
		woStatePOU := 10;
		boDonePOU := FALSE;
	ELSIF R_TRIG_Start.Q THEN
		woStatePOU := 1;
		boDonePOU := FALSE;
	END_IF;
	
	1:	//Running

	IF boErrorPOU THEN
		woStatePOU := 10;
	ELSIF R_TRIG_Start.Q THEN
		woStatePOU := 10;	 
		boErrorTransitionLST := TRUE;
	ELSIF R_TRIG_Stop.Q THEN
		woStatePOU := 2;
	ELSIF R_TRIG_Done.Q THEN
		woStatePOU := 2;
		boDonePOU := TRUE;
	END_IF;
	
	2:	//Stopping

	IF boErrorPOU THEN
		woStatePOU := 10;
	ELSIF R_TRIG_Start.Q THEN
		boErrorTransitionLST := TRUE;
		woStatePOU := 10;
	ELSIF regAsycubeReadPIO.HR_MODBUS_SEQUENCE_STATUS.w = 0 THEN
		woStatePOU := 0;
	END_IF;
	
	10:	//Error

	IF NOT boErrorPOU THEN
		woStatePOU := 2;
	END_IF;
	
END_CASE;

//Parameters processing

//If it is in IDLE
IF woStatePOU = 0 THEN
	regAsycubeWritePIO.HR_SEQUENCE_HALT.w := 0;
END_IF;

//If it is in running (trigger)
IF R_TRIG_State1.Q THEN
	regAsycubeWritePIO.HR_SEQUENCE_EXECUTION_TRIG.w := 1;
END_IF;

//If it is in stopping
IF woStatePOU = 2 THEN
	regAsycubeWritePIO.HR_SEQUENCE_EXECUTION_TRIG.w := 0;
	regAsycubeWritePIO.HR_SEQUENCE_HALT.w := 1;
	regAsycubeWritePIO.HR_MODBUS_CONTROL.w := 16#00;
END_IF;
	 
//If it is in error
IF woStatePOU = 10 THEN
	regAsycubeWritePIO.HR_SEQUENCE_EXECUTION_TRIG.w := 0;
	regAsycubeWritePIO.HR_SEQUENCE_HALT.w := 1;
END_IF;

//Save last state before error state
IF woStatePOU <> 10 THEN
	woLastStateLST := woStatePOU;
END_IF;

//If it is in error (trigger)
IF (R_TRIG_Stop.Q AND woStatePOU = 10) OR 
	((regAsycubeReadPIO.HR_MODBUS_COMMUNICATION_STATUS_L.w = 4 AND regAsycubeReadPIO.HR_ETHERCAT_COMMUNICATION_STATUS.w = 8) AND 
	(boErrorComAsycubeLST OR boErrorComGatewayLST) AND 
	woLastStateLST = 0) THEN
	
	regAsycubeWritePIO.HR_MODBUS_CONTROL.w := 16#FF;
	boErrorTransitionLST := FALSE;
	boErrorTimeOutLST := FALSE;
	boErrorComAsycubeLST := FALSE;
	boErrorComGatewayLST := FALSE;
	boErrorParameterLST := FALSE;
END_IF;

//Affectation of paramters for axis X
IF inXPosPIN > 100 AND woStatePOU = 1 THEN
	boErrorParameterLST := TRUE;
ELSIF inXPosPIN < -100 AND woStatePOU = 1 THEN
	boErrorParameterLST := TRUE;
ELSIF woStatePOU = 1 THEN
	regAsycubeWritePIO.HR_SEQUENCE_EXECUTION_X.w := inXPosPIN;
END_IF;

//Affectation of paramters for axis Y
IF inYPosPIN > 100  AND woStatePOU = 1 THEN
	boErrorParameterLST := TRUE;
ELSIF inYPosPIN < -100 AND woStatePOU = 1 THEN
	boErrorParameterLST := TRUE;
ELSIF woStatePOU = 1 THEN
	regAsycubeWritePIO.HR_SEQUENCE_EXECUTION_Y.w := inYPosPIN;
END_IF;
	 
//Write another parameters
regAsycubeWritePIO.HR_SEQUENCE_EXECUTION_NBMAX.w := inNbPartsMaxPIN;
regAsycubeWritePIO.HR_SEQUENCE_EXECUTION_NBPARTS.w := inNbPartsPIN;

//Sequence ID parameter
IF inSeqIDPIN > 26 AND woStatePOU = 1 THEN
	boErrorParameterLST := TRUE;
ELSIF inSeqIDPIN < 1 AND woStatePOU = 1 THEN
	boErrorParameterLST := TRUE;
ELSIF woStatePOU = 1 THEN
	regAsycubeWritePIO.HR_SEQUENCE_EXECUTION_SEQUENCEID.w := inSeqIDPIN;
END_IF;

//Vibration set parameter
IF inVibrationSetPIN > 26 AND woStatePOU = 1 THEN
	boErrorParameterLST := TRUE;
ELSIF inVibrationSetPIN < 1 AND woStatePOU = 1 THEN
	boErrorParameterLST := TRUE;	 
ELSIF woStatePOU = 1 THEN
	regAsycubeWritePIO.HR_SELECT_VIBRATION_SET.w := inVibrationSetPIN;
END_IF;
		  
//Time remaining
tiRemainingTimePOU := INT_TO_TIME(regAsycubeReadPIO.HR_SEQUENCE_REMAINING_TIME.w);
		  
{endregion}

//Management of backlight 
{region "Backlight"}

//Turn ON or OFF the backlight
regAsycubeWritePIO.HR_BACKLIGHT_STATE_CONTROL.w := BOOL_TO_INT(boBacklightPIN AND woStatePOU <> 10);

//State of backlight
boBacklightStatePOU := INT_TO_BOOL(regAsycubeReadPIO.HR_BACKLIGHT_STATE_STATUS.w);

{endregion}

//Management of error
{region "Error"}
	
//Time out communciation	
IF TON_TimeOut.Q THEN
	boErrorTimeOutLST := TRUE;
END_IF;

//Asycube disconnected
IF regAsycubeReadPIO.HR_MODBUS_COMMUNICATION_STATUS_L.w <> 4 AND woStatePOU <> 10 THEN
	boErrorComAsycubeLST := TRUE;
END_IF;

//Gateway disconnected
IF regAsycubeReadPIO.HR_ETHERCAT_COMMUNICATION_STATUS.w <> 8 AND woStatePOU <> 10 THEN
	boErrorComGatewayLST := TRUE;
END_IF;
  
//If an error is active
IF	((regAsycubeReadPIO.HR_MODBUS_STATUS.w <> 0 OR boErrorTransitionLST OR boErrorParameterLST) AND woStatePOU <> 0) OR 
	(woStatePOU = 0 AND (INT_TO_UINT(regAsycubeReadPIO.HR_ALARMS.w) AND 16#40) = 16#40) 
	OR boErrorTimeOutLST OR regAsycubeReadPIO.HR_MODBUS_SEQUENCE_STATUS.w = 2 
	OR boErrorComAsycubeLST OR boErrorComGatewayLST THEN
		 
	boErrorPOU := TRUE;
			
		//Error transition
		IF boErrorTransitionLST THEN
			inErrorIDPOU := 700;
			stErrorNamePOU := 'Transition Error';
		//Asycube  Modbus  errors  status
		ELSIF (INT_TO_UINT(regAsycubeReadPIO.HR_MODBUS_STATUS.w) AND 16#01) = 16#01 THEN	
			inErrorIDPOU := 701;	
	  		stErrorNamePOU := 'Asycube Modbus Error : 0x';
			stErrorNamePOU := CONCAT(STR1:= stErrorNamePOU, STR2:= DWORD_TO_HEXSTR( UINT_TO_DWORD( INT_TO_UINT(regAsycubeReadPIO.HR_MODBUS_ERROR_CODE.w) AND 16#00FF ), 4, FALSE ) ); 
				 
		//Internal  Modbus  communication  errorstatus
		ELSIF (INT_TO_UINT(regAsycubeReadPIO.HR_MODBUS_STATUS.w) AND 16#02) = 16#02 THEN
			inErrorIDPOU := 702;
			stErrorNamePOU := 'Asycube Internal Modbus Error : 0x';
			stErrorNamePOU := CONCAT(STR1:= stErrorNamePOU, STR2:= DWORD_TO_HEXSTR( UINT_TO_DWORD( SHL( INT_TO_UINT(regAsycubeReadPIO.HR_MODBUS_ERROR_CODE.w) AND 16#FF00 , 2) ) , 4, FALSE ) ); 
						   
		//Asycube  warnings  status
		ELSIF (INT_TO_UINT(regAsycubeReadPIO.HR_MODBUS_STATUS.w) AND 16#04) = 16#04 THEN
			inErrorIDPOU := 703;
			stErrorNamePOU := 'Asycube Warnings : 0x';
			stErrorNamePOU := CONCAT(STR1:= stErrorNamePOU, STR2:= DWORD_TO_HEXSTR( INT_TO_DWORD(regAsycubeReadPIO.HR_WARNINGS.w), 4, FALSE ) ); 

		//Asycube alarms status
		ELSIF (INT_TO_UINT(regAsycubeReadPIO.HR_MODBUS_STATUS.w) AND 16#08) = 16#08 THEN
			inErrorIDPOU := 704;
			stErrorNamePOU := 'Asycube Alarms : 0x';
			stErrorNamePOU := CONCAT(STR1:= stErrorNamePOU, STR2:= DWORD_TO_HEXSTR( INT_TO_DWORD(regAsycubeReadPIO.HR_ALARMS.w), 4, FALSE ) );   	
 		
		//Gateway disconnected from plc
		ELSIF boErrorComGatewayLST THEN
			inErrorIDPOU := 705;
			stErrorNamePOU := 'Gateway disconnected from PLC';
		
		//Asycube disconnected from gateway
		ELSIF boErrorComAsycubeLST THEN
			inErrorIDPOU := 706;
			stErrorNamePOU := 'Asycube disconnected from gateway';
		
		//Communication time out
		ELSIF boErrorTimeOutLST THEN
			inErrorIDPOU := 707;
			stErrorNamePOU := 'Time out';
			 
		//Incorrect parameters
		ELSIF boErrorParameterLST THEN
			inErrorIDPOU := 708;
			stErrorNamePOU := 'Wrong parameter';
			//See variable error
			IF inXPosPIN > 100 OR inXPosPIN < -100 THEN
				stErrorNamePOU := CONCAT(stErrorNamePOU , ' : inXPosPIN' );
			ELSIF inYPosPIN > 100 OR inYPosPIN < -100 THEN
				stErrorNamePOU := CONCAT(stErrorNamePOU , ' : inYPosPIN' );
			ELSIF inSeqIDPIN > 26 OR inSeqIDPIN < 1 THEN
				stErrorNamePOU := CONCAT(stErrorNamePOU , ' : inSeqIDPIN' );
			ELSIF inVibrationSetPIN > 26 OR inVibrationSetPIN < 1 THEN
				stErrorNamePOU := CONCAT(stErrorNamePOU , ' : inVibrationSetPIN' );
			END_IF;
			
		//Unknown error	 
		ELSE 
			inErrorIDPOU := 709;
			stErrorNamePOU := 'N/A';
		END_IF;  

ELSE
	boErrorPOU := FALSE;
	inErrorIDPOU := 0;
	stErrorNamePOU := '';	 
END_IF;

{endregion}

END_FUNCTION_BLOCK

// POUs/MAIN
PROGRAM MAIN
VAR
	FB_Sequence_0					: FB_Execute_Sequence;
	FB_Platform_0					: FB_Execute_Platform_Vibration;
	FB_Hopper_0						: FB_Execute_Hopper_Vibration;
	FB_Backlight_0					: FB_Backlight;
	
	boStartSeqLST: BOOL;
	boStopSeqLST: BOOL;
	inSeqIDLST: INT;
	inVibrationIDSeqLST: INT;
	inNbPartSeqLST: INT;
	inNbPartMaxSeqLST: INT;
	inPartPositionXLST: INT;
	inPartPositionYLST: INT;
	boBacklightSeqLST: BOOL;
	inSelectModePlatformLST: INT;
	boStartPlatformLST: BOOL;
	boStopPlatformLST: BOOL;
	inVibrationIDPlatformLST: INT;
	tiDurationPlatformLST: TIME := T#1S;
	inSelectModeHopperLST: INT;
	boStartHopperLST: BOOL;
	boStopHopperLST: BOOL;
	inVibrationIDHopperLST: INT;
	inNbPartHopperLST: INT;
	inNbPartMaxHopperLST: INT;
	tiDurationHopperLST: TIME := T#1S;
	boLightONLST: BOOL;
	tuDurationLightLST: TIME := T#1S;
	boLightOFFLST: BOOL;

END_VAR

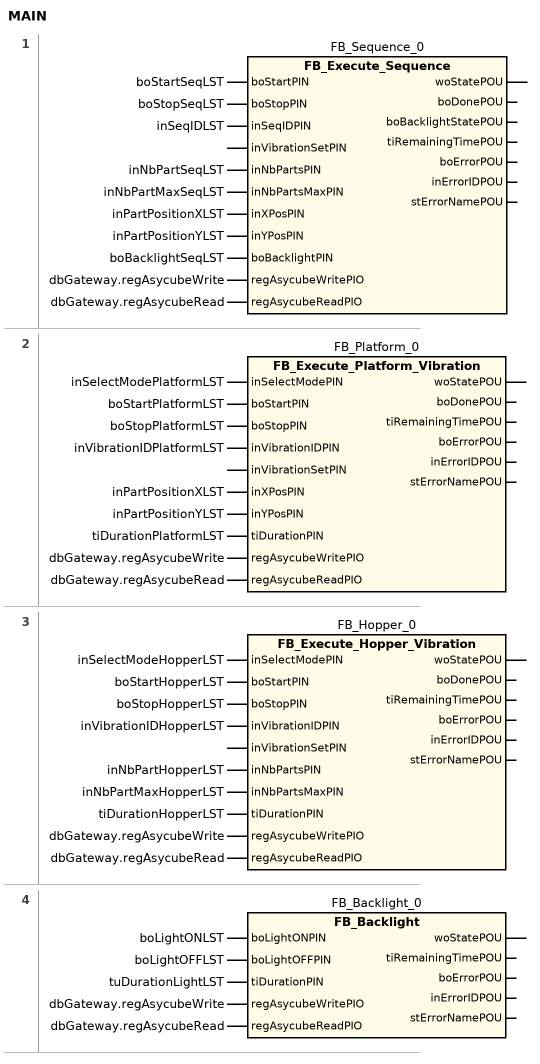
// NETWORK 1
FB_Sequence_0(
    boStartPIN := boStartSeqLST,
    boStopPIN := boStopSeqLST,
    inSeqIDPIN := inSeqIDLST,
    inNbPartsPIN := inNbPartSeqLST,
    inNbPartsMaxPIN := inNbPartMaxSeqLST,
    inXPosPIN := inPartPositionXLST,
    inYPosPIN := inPartPositionYLST,
    boBacklightPIN := boBacklightSeqLST,
    regAsycubeWritePIO := dbGateway.regAsycubeWrite,
    regAsycubeReadPIO := dbGateway.regAsycubeRead); // FB_Execute_Sequence

// NETWORK 2
FB_Platform_0(
    inSelectModePIN := inSelectModePlatformLST,
    boStartPIN := boStartPlatformLST,
    boStopPIN := boStopPlatformLST,
    inVibrationIDPIN := inVibrationIDPlatformLST,
    inXPosPIN := inPartPositionXLST,
    inYPosPIN := inPartPositionYLST,
    tiDurationPIN := tiDurationPlatformLST,
    regAsycubeWritePIO := dbGateway.regAsycubeWrite,
    regAsycubeReadPIO := dbGateway.regAsycubeRead); // FB_Execute_Platform_Vibration

// NETWORK 3
FB_Hopper_0(
    inSelectModePIN := inSelectModeHopperLST,
    boStartPIN := boStartHopperLST,
    boStopPIN := boStopHopperLST,
    inVibrationIDPIN := inVibrationIDHopperLST,
    inNbPartsPIN := inNbPartHopperLST,
    inNbPartsMaxPIN := inNbPartMaxHopperLST,
    tiDurationPIN := tiDurationHopperLST,
    regAsycubeWritePIO := dbGateway.regAsycubeWrite,
    regAsycubeReadPIO := dbGateway.regAsycubeRead); // FB_Execute_Hopper_Vibration

// NETWORK 4
FB_Backlight_0(
    boLightONPIN := boLightONLST,
    boLightOFFPIN := boLightOFFLST,
    tiDurationPIN := tuDurationLightLST,
    regAsycubeWritePIO := dbGateway.regAsycubeWrite,
    regAsycubeReadPIO := dbGateway.regAsycubeRead); // FB_Backlight

END_PROGRAM
